SUBAPPLICATION Uebung_019c (* Umschalten einer Maske *)
  (* Standard: 61499-2; Description: Copyright (c) 2023 Meisterschulen am Ostbahnhof This program and the accompanying materials are made available under the terms of the Eclipse Public License 2.0 which is available at https://www.eclipse.org/legal/epl-2.0/ SPDX-License-Identifier: EPL-2.0 *)
  (* Version 1.0, 2023-10-23, Franz Höpfinger, Meisterschulen am Ostbahnhof, initial API and implementation and/or initial documentation *)
  PACKAGE Uebungen;
  IMPORT Uebungen::const::UT::DefaultPool::AlarmMask_A2_medium;
  IMPORT Uebungen::const::UT::DefaultPool::DataMask_M1;
  IMPORT Uebungen::const::UT::DefaultPool::DataMask_M2;
  IMPORT logiBUS::io::DI::logiBUS_DI::Input_I1;
  IMPORT logiBUS::io::DI::logiBUS_DI::Input_I2;
  IMPORT logiBUS::io::DI::logiBUS_DI::Input_I3;
  IMPORT logiBUS::io::DI::logiBUS_DI::Input_I4;
  IMPORT logiBUS::io::DI::logiBUS_DI_Events::BUTTON_SINGLE_CLICK;
  IMPORT logiBUS::io::DQ::logiBUS_DO::Output_Q8;
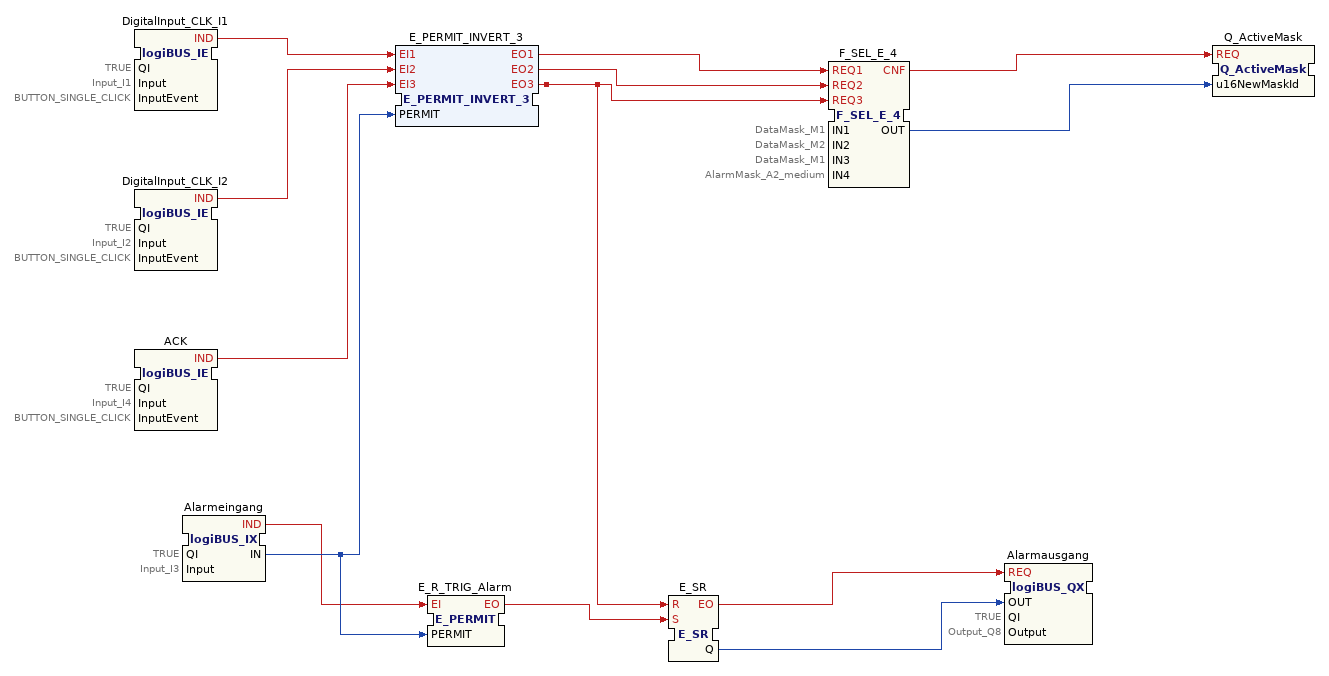
  FBS
    DigitalInput_CLK_I1 : logiBUS::io::DI::logiBUS_IE(QI := TRUE, Input := Input_I1, InputEvent := BUTTON_SINGLE_CLICK);
    Q_ActiveMask : isobus::UT::Q::Q_ActiveMask;
    DigitalInput_CLK_I2 : logiBUS::io::DI::logiBUS_IE(QI := TRUE, Input := Input_I2, InputEvent := BUTTON_SINGLE_CLICK);
    F_SEL_E_4 : eclipse4diac::utils::selection::F_SEL_E_4(IN1 := DataMask_M1, IN2 := DataMask_M2, IN3 := DataMask_M1, IN4 := AlarmMask_A2_medium);
    ACK : logiBUS::io::DI::logiBUS_IE(QI := TRUE, Input := Input_I4, InputEvent := BUTTON_SINGLE_CLICK);
    E_SR : iec61499::events::E_SR;
    Alarmausgang : logiBUS::io::DQ::logiBUS_QX(QI := TRUE, Output := Output_Q8);
    Alarmeingang : logiBUS::io::DI::logiBUS_IX(QI := TRUE, Input := Input_I3);
    E_R_TRIG_Alarm : iec61499::events::E_PERMIT;
  END_FBS
  SUBAPPS
    E_PERMIT_INVERT_3 : MyLib::sys::E_PERMIT_INVERT_3;
  END_SUBAPPS
  EVENT_CONNECTIONS
    F_SEL_E_4.CNF TO Q_ActiveMask.REQ;
    DigitalInput_CLK_I1.IND TO E_PERMIT_INVERT_3.EI1;
    E_PERMIT_INVERT_3.EO1 TO F_SEL_E_4.REQ1;
    DigitalInput_CLK_I2.IND TO E_PERMIT_INVERT_3.EI2;
    E_PERMIT_INVERT_3.EO2 TO F_SEL_E_4.REQ2;
    ACK.IND TO E_PERMIT_INVERT_3.EI3;
    E_PERMIT_INVERT_3.EO3 TO F_SEL_E_4.REQ3;
    E_PERMIT_INVERT_3.EO3 TO E_SR.R;
    E_SR.EO TO Alarmausgang.REQ;
    Alarmeingang.IND TO E_R_TRIG_Alarm.EI;
    E_R_TRIG_Alarm.EO TO E_SR.S;
  END_CONNECTIONS
  DATA_CONNECTIONS
    F_SEL_E_4.OUT TO Q_ActiveMask.u16NewMaskId;
    E_SR.Q TO Alarmausgang.OUT;
    Alarmeingang.IN TO E_R_TRIG_Alarm.PERMIT;
    Alarmeingang.IN TO E_PERMIT_INVERT_3.PERMIT;
  END_CONNECTIONS
END_SUBAPPLICATION
